GLOBALCONSTANTS IG3_Source_Addresses (* Industry Group 3 specific source addresses *)
  (* Standard: 61499-1 *)
  (* Version 1.0, 2026-06-29, Franz Höpfinger, Demmler Andreas Fahrzeugbau *)
  PACKAGE isobus::pgn::const;
  VAR_GLOBAL CONSTANT
    SA_RESERVED_128 : BYTE := 128; (* Source Address: thru 207 are reserved for future assignment by SAE - Used for dynamic address *)
    SA_RESERVED_208 : BYTE := 208; (* Source Address: thru 223 are reserved for future assignment - Used for individual preassigned *)
    SA_ROTATION_SENSOR : BYTE := 224; (* Source Address: Rotation Sensor - A device that measures the rotational angle around an axis. *)
    SA_LIFT_ARM_CONTROLLER : BYTE := 225; (* Source Address: Lift Arm Controller - Controls the lift arms and tilt functions on a construction *)
    SA_SLOPE_SENSOR : BYTE := 226; (* Source Address: Slope Sensor - A device that measures the slope along an axis. *)
    SA_MAIN_CONTROLLER_SKID_STEER_LOADER : BYTE := 227; (* Source Address: Main Controller - Skid Steer Loader - Primary system controller for skid steer *)
    SA_LOADER_CONTROL : BYTE := 228; (* Source Address: Loader Control - Controls the hydraulic system of the loader attachment of a *)
    SA_LASER_TRACER : BYTE := 229; (* Source Address: Laser Tracer - A device that receives a laser strike and reports the vertical and *)
    SA_LAND_LEVELING_SYSTEM_DISPLAY : BYTE := 230; (* Source Address: Land Leveling System Display - This device displays position information at a *)
    SA_SINGLE_LAND_LEVELING_SYSTEM_SUPERVISOR : BYTE := 231; (* Source Address: Single Land Leveling System Supervisor - This device is the Land Leveling System *)
    SA_LAND_LEVELING_ELECTRIC_MAST : BYTE := 232; (* Source Address: Land Leveling Electric Mast - A device that moves a Sensor to maintain a specific *)
    SA_SINGLE_LAND_LEVELING_SYSTEM_OPERATOR_INTERFACE : BYTE := 233; (* Source Address: Single Land Leveling System Operator Interface - A component that allows the user *)
    SA_LASER_RECEIVER : BYTE := 234; (* Source Address: Laser Receiver - A device that receives a laser strike, and reports the specific *)
    SA_SUPPLEMENTAL_SENSOR_PROCESSING_UNIT_1 : BYTE := 235; (* Source Address: Supplemental Sensor Processing Unit #1 *)
    SA_SUPPLEMENTAL_SENSOR_PROCESSING_UNIT_2 : BYTE := 236; (* Source Address: Supplemental Sensor Processing Unit #2 *)
    SA_SUPPLEMENTAL_SENSOR_PROCESSING_UNIT_3 : BYTE := 237; (* Source Address: Supplemental Sensor Processing Unit #3 *)
    SA_SUPPLEMENTAL_SENSOR_PROCESSING_UNIT_4 : BYTE := 238; (* Source Address: Supplemental Sensor Processing Unit #4 *)
    SA_SUPPLEMENTAL_SENSOR_PROCESSING_UNIT_5 : BYTE := 239; (* Source Address: Supplemental Sensor Processing Unit #5 *)
    SA_SUPPLEMENTAL_SENSOR_PROCESSING_UNIT_6 : BYTE := 240; (* Source Address: Supplemental Sensor Processing Unit #6 *)
    SA_ENGINE_MONITOR_1 : BYTE := 241; (* Source Address: Engine Monitor #1 *)
    SA_ENGINE_MONITOR_2 : BYTE := 242; (* Source Address: Engine Monitor #2 *)
    SA_ENGINE_MONITOR_3 : BYTE := 243; (* Source Address: Engine Monitor #3 *)
    SA_ENGINE_MONITOR_4 : BYTE := 244; (* Source Address: Engine Monitor #4 *)
    SA_ENGINE_MONITOR_5 : BYTE := 245; (* Source Address: Engine Monitor #5 *)
    SA_ENGINE_MONITOR_6 : BYTE := 246; (* Source Address: Engine Monitor #6 *)
    SA_ENGINE_MONITOR_7 : BYTE := 247; (* Source Address: Engine Monitor #7 *)
  END_VAR
END_GLOBALCONSTANTS
